TYPE ARCommunicationSendPacketValue :
STRUCT
END_STRUCT
	key : STRING(255), // key for accsessiong the data
	as : ARCommunicationSendPacketValueStore_t, // union for storing the data
	valueType : ARCommunicationValueType_t // safes value type
END_TYPE

(* stored: Version 1.1.0.1
   DUT ARCommunicationSendPacketValue: Id {b76ecd42-be41-4c52-839a-229d481633d2} *)
